# EPICS substitutions: DPU08/DPU08.substitutions
file "/usr/local/epics/asyn4-29/db/asynRecord.db" { pattern
{P,           R,       PORT,      ADDR,   IMAX,    OMAX}
{TMSR:,    DCS,    DPU08,     0,      80,      80}
}
file "../../db/statistics.template" { pattern
{P,           R,         PORT,          SCAN}
}
